FUNCTION_BLOCK FB_2CAM_CameraSequenceNo
VAR_INPUT
	aCameraTrigger		: ARRAY[0..6] OF BOOL;
END_VAR
VAR_OUTPUT
	nCamera1ScanNo		: INT;
	nCamera2ScanNo		: INT;
END_VAR
VAR
END_VAR

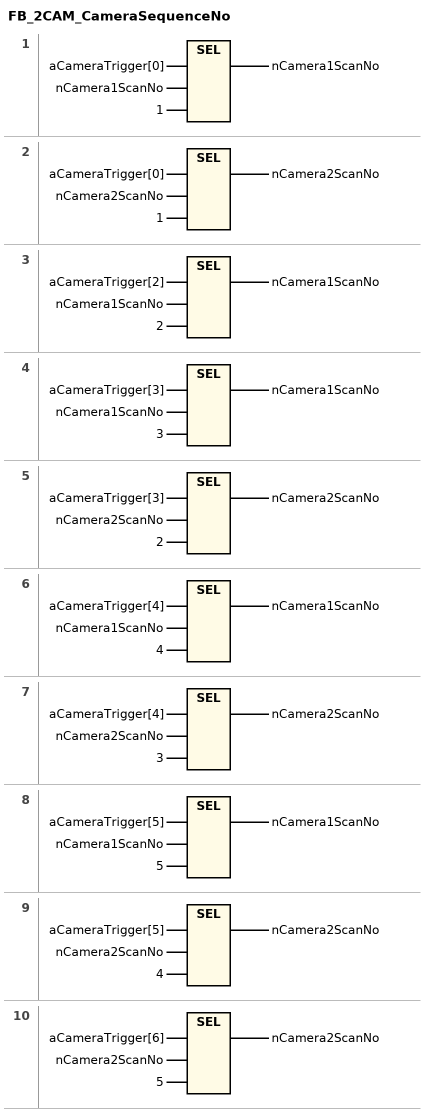
// NETWORK 1
nCamera1ScanNo := SEL(aCameraTrigger[0], nCamera1ScanNo, 1);

// NETWORK 2
nCamera2ScanNo := SEL(aCameraTrigger[0], nCamera2ScanNo, 1);

// NETWORK 3
nCamera1ScanNo := SEL(aCameraTrigger[2], nCamera1ScanNo, 2);

// NETWORK 4
nCamera1ScanNo := SEL(aCameraTrigger[3], nCamera1ScanNo, 3);

// NETWORK 5
nCamera2ScanNo := SEL(aCameraTrigger[3], nCamera2ScanNo, 2);

// NETWORK 6
nCamera1ScanNo := SEL(aCameraTrigger[4], nCamera1ScanNo, 4);

// NETWORK 7
nCamera2ScanNo := SEL(aCameraTrigger[4], nCamera2ScanNo, 3);

// NETWORK 8
nCamera1ScanNo := SEL(aCameraTrigger[5], nCamera1ScanNo, 5);

// NETWORK 9
nCamera2ScanNo := SEL(aCameraTrigger[5], nCamera2ScanNo, 4);

// NETWORK 10
nCamera2ScanNo := SEL(aCameraTrigger[6], nCamera2ScanNo, 5);

END_FUNCTION_BLOCK

(* stored: Version 1.1.0.1, ProductVersion 3.1.4024.15
   POU FB_2CAM_CameraSequenceNo: Id {ca8d559a-e744-4260-ae43-85083ef61da2}, SpecialFunc None *)
